TYPE ST_ArrayProperties :
STRUCT
	Count		: DINT;
	StartIndex	: T_ArrayIndexer;
	EndIndex	: T_ArrayIndexer;
END_STRUCT
END_TYPE

(* stored: Version 1.1.0.1, ProductVersion 3.1.4024.14
   DUT ST_ArrayProperties: Id {b1c37182-4802-057e-1db3-4f1525616de3} *)
